//==================================================================================================
//							Beckhoff Automation Poland
//									12.04.2018
//	Blok funkcyjny kontroli luzownika w silniku podpietym do AX8000. Przewaga ForceLock
//	Dzialania na obiekcie: 3000:07 Motor brake force
//	Index:			AxisMainSlot: 16#3000 (Ch A)/ 16#3400 (Ch B)
//	Subindex:		16#07
//	Datatype:		ENUM (INT16)
//	Enum Value:		0 (0x00): 	Release_force
//					1 (0x01): 	Force_lock
//					2 (0x02): 	Force_unlock
//
//  v1.0	|| TC v 3.1.4022.16		|| - pierwsza wersja
//==================================================================================================
FUNCTION_BLOCK FB_HoldingBrakeCtrlAX8000
VAR_INPUT
	bForceLock 						: BOOL;								// 
	bForceUnlock					: BOOL;								// 
	stDriveRef						: ST_DriveRef;
END_VAR
VAR_OUTPUT
	bBusy							: BOOL;
	bError							: BOOL; 							// General error: parameter or CoE read.
																		// If bError = TRUE and bInitialized = FALSE - error during read motor data.
																		// If bError = TRUE and bInitialized = TRUE and (iAdsErrId <> 0 or iCANopenErrId <> 0) then I2T read error
																		// If bError = TRUE and bInitialized = TRUE and iAdsErrId = 0 and iCANopenErrId = 0 then parameter error: rTorqueLimit outside permitted range rTorqueLimitLow..rTorqueLimitHigh or Empty stDriveRef
	iAdsErrId						: UINT;								// Forwarded output FB_CoERead_ByDriveRef
	iCANopenErrId					: UINT;								// Forwarded output FB_CoERead_ByDriveRef
END_VAR
VAR
	bExecute						: BOOL;
	iMotorBrakeForce				: INT;								// 0 - Release_force, 1 - Force_lock, 2 - Force_unlock
	rtForceLock						: R_TRIG;
	rtForceUnlock					: R_TRIG;
	ftForceLock						: F_TRIG;
	ftForceUnlock					: F_TRIG;
	fbForceLockUnlock				: FB_CoEWrite_ByDriveRef;
END_VAR

{region "Call triggers"}
//======================= Call triggers =========================
rtForceLock(CLK:= bForceLock);
ftForceLock(CLK:= bForceLock);
rtForceUnlock(CLK:= bForceUnlock);
ftForceUnlock(CLK:= bForceUnlock);
bExecute								:= rtForceLock.Q OR ftForceLock.Q OR rtForceUnlock.Q OR ftForceUnlock.Q;
//===============================================================
{endregion}
{region "Main code"}
//========================= Main code ===========================
IF bExecute THEN
	iMotorBrakeForce 						:= 0;										// Clear value
	iMotorBrakeForce.1 						:= bForceUnlock;							// Set force unlock bit
	iMotorBrakeForce 						:= SEL(bForceLock, iMotorBrakeForce, 1);	// Set force lock bit, it has higher priority than unlock
END_IF

fbForceLockUnlock(	stDriveRef				:= stDriveRef, 
					nIndex					:= 16#3000 + (stDriveRef.nDriveNo * 16#400), 
					nSubIndex				:= 16#07, 
					pSrcBuf					:= ADR(iMotorBrakeForce), 
					cbBufLen				:= SIZEOF(iMotorBrakeForce), 
					bExecute				:= bExecute,
					bBusy					=> bBusy, 
					bError					=> bError, 
					iAdsErrId				=> iAdsErrId, 
					iCANopenErrId			=> iCANopenErrId);
//===============================================================
{endregion}

END_FUNCTION_BLOCK

(* stored: Version 1.1.0.1, ProductVersion 3.1.4026.13, FileIdentifier f1a6c7ed213e233c69bca35558d0f6f85ace7af8, FileSignature 2e62a2bec5752900292b47057b8f6394ef24ad61f2d796daf3b47aef7c38555b6838c428d88ef1a0529522c33d8e6850c19f43a5b3dfaa7b75468c1764140818e03a62888fda451656ea431d0eea525dd8ae64999d8a2982e35380499d8a53335001069e8dc8a304c96b1a77e1de38da9d4ead6d59e4ac5b76a636fb8dcfddb04d587b084efc06d57b1a670d3e6e82c718cecaa342e2b5010d8f6515c06b4edce70c57f2de41e3412a3f1e5b8ae1f162d48da0449704c8394c54a90a04a9c716e6361fcd0d0758d015141fa4bcc22b43026d314e41aaff81a2fff6d913bf0cf6c643660994863c1654010251cbf1a893700b6b8532e3fee7f6972d0f9d46924e
   POU FB_HoldingBrakeCtrlAX8000: Id {53f74e01-16e6-4f84-b28b-e957b293a916}, SpecialFunc None *)
